// TwinCAT 3 PLC project PLC_TMO_VAC
// ProgramVersion: 3.1.4022.7
// libraries:
//   LCLS General, * (SLAC)
//   LCLS Vacuum, * (SLAC - LCLS)
//   PMPS, * (SLAC - LCLS)
//   Tc2_Standard, * (Beckhoff Automation GmbH)
//   Tc2_System, * (Beckhoff Automation GmbH)
//   Tc3_Module, * (Beckhoff Automation GmbH)
// project tree:
//   GVLs/ GVL_FEE_Device.TcGVL, GVL_PMPS.TcGVL, GVL_Variables.TcGVL
//   / PlcTask.TcTTO
//   POUs/ DIAGNOSTICS.TcPOU, MAIN.TcPOU, PRG_FEE.TcPOU, PRG_Section_2.TcPOU
// real-time tasks:
//   TASK PlcTask: cycle T#10ms, priority 20, ADS port 350
// I/O:
//   DEVICE Device 1 (EtherCAT), AmsNetId 5.59.117.180.2.1
//     B940-R20-CX0 (EK1200) [EK1200-5000 EtherCAT Power supply (2A E-Bus)]
//       CX0_E1 (EL2202)
//       CX0_E2 (EL1008)
//       CX0_E3 (EL2008)
//       CX0_E4 (EL2794)
//       CX0_E5 (EL6070)
//       CX0_E6_QPC1 (EL3064)
//       CX0_E7_QPC1 (EL1004)
//       CX0_E8_QPC1 (EL2794)
//       CX0_E9_QPC2 (EL3064)
//       CX0_E10_QPC2 (EL1004)
//       CX0_E11_QPC2 (EL2794)
//       CX0_E12 (EL6001)
//       EK1122-0080
//       EK (EL6692) [EL6692 EtherCAT Bridge terminal (Primary)]
//       CX0_EK1110
//     B940_R20_EK0 (EK1100) [EK1100 EtherCAT Coupler (2A E-Bus)]
//       Term 41 (EL3064)
//       Term 42 (EL3064)
//       Term 43 (EL2794)
//       Term 44 (EL9505)
//       Term 45 (EL1124)
//       Term 46 (EK1110)
//     B940_K4S20_EK0  (EK1100) [EK1100 EtherCAT Coupler (2A E-Bus)]
//       K420-E1-FSV (EL1004)
//       K420-E2-FSV (EL2202)
//       K420-E13-FSV (EL2202)
//       K420-E4-FSV (EK1110)
//     B940_K4S20_EB1  (EP2338-0002)
//     B940_K4S20_EB2  (EP3174-0002)
//     B940_K4S20_EB3 (EP2624-0002)
//     B940_K4S24_EB1 (EP3174-0002)
//     B940_K4S24_EB2 (EP2624-0002)
//     B940_K4S28_EB1 (EP3174-0002)
//     B940_K4S28_EB2 (EP2624-0002)
//     B940_K4S33_EB1 (EP2338-0002)
//     B940_K4S33_EB2 (EP3174-0002)
//     B940_K4S33_EB3 (EP2624-0002)
// variable links:
//   PLC_TMO_VAC Instance <-> Device 1 (EtherCAT)/B940-R20-CX0 (EK1200)/CX0_E10_QPC2 (EL1004)
//     PlcTask Inputs/GVL_FEE_Device.PC4K4_XTES_PIP_01.i_xSP_DI <-> Channel 1/Input
//   PLC_TMO_VAC Instance <-> Device 1 (EtherCAT)/B940-R20-CX0 (EK1200)/CX0_E11_QPC2 (EL2794)
//     PlcTask Outputs/GVL_FEE_Device.PC4K4_XTES_PIP_01.q_xHVEna_DO <-> Channel 1/Output
//   PLC_TMO_VAC Instance <-> Device 1 (EtherCAT)/B940-R20-CX0 (EK1200)/CX0_E6_QPC1 (EL3064)
//     PlcTask Inputs/GVL_FEE_Device.MR1K4_SOMS_PIP_01.i_iPRESS <-> AI Standard Channel 1/Value
//     PlcTask Inputs/GVL_FEE_Device.ST1K4_TEST_PIP_01.i_iPRESS <-> AI Standard Channel 2/Value
//     PlcTask Inputs/GVL_FEE_Device.ST2K4_BCS_PIP_01.i_iPRESS <-> AI Standard Channel 3/Value
//     PlcTask Inputs/GVL_FEE_Device.ST3K4_PPS_PIP_01.i_iPRESS <-> AI Standard Channel 4/Value
//   PLC_TMO_VAC Instance <-> Device 1 (EtherCAT)/B940-R20-CX0 (EK1200)/CX0_E7_QPC1 (EL1004)
//     PlcTask Inputs/GVL_FEE_Device.MR1K4_SOMS_PIP_01.i_xSP_DI <-> Channel 1/Input
//     PlcTask Inputs/GVL_FEE_Device.ST1K4_TEST_PIP_01.i_xSP_DI <-> Channel 2/Input
//     PlcTask Inputs/GVL_FEE_Device.ST2K4_BCS_PIP_01.i_xSP_DI <-> Channel 3/Input
//     PlcTask Inputs/GVL_FEE_Device.ST3K4_PPS_PIP_01.i_xSP_DI <-> Channel 4/Input
//   PLC_TMO_VAC Instance <-> Device 1 (EtherCAT)/B940-R20-CX0 (EK1200)/CX0_E8_QPC1 (EL2794)
//     PlcTask Outputs/GVL_FEE_Device.MR1K4_SOMS_PIP_01.q_xHVEna_DO <-> Channel 1/Output
//     PlcTask Outputs/GVL_FEE_Device.ST1K4_TEST_PIP_01.q_xHVEna_DO <-> Channel 2/Output
//     PlcTask Outputs/GVL_FEE_Device.ST2K4_BCS_PIP_01.q_xHVEna_DO <-> Channel 3/Output
//     PlcTask Outputs/GVL_FEE_Device.ST3K4_PPS_PIP_01.q_xHVEna_DO <-> Channel 4/Output
//   PLC_TMO_VAC Instance <-> Device 1 (EtherCAT)/B940-R20-CX0 (EK1200)/CX0_E9_QPC2 (EL3064)
//     PlcTask Inputs/GVL_FEE_Device.PC4K4_XTES_PIP_01.i_iPRESS <-> AI Standard Channel 1/Value
//   PLC_TMO_VAC Instance <-> Device 1 (EtherCAT)/B940_K4S20_EB1  (EP2338-0002)
//     PlcTask Inputs/GVL_FEE_Device.TV1K4_VGC_01.i_xClsLS <-> Channel 2/Input
//     PlcTask Inputs/GVL_FEE_Device.TV1K4_VGC_02.i_xClsLS <-> Channel 6/Input
//     PlcTask Inputs/GVL_FEE_Device.TV1K4_VGC_01.i_xOpnLS <-> Channel 1/Input
//     PlcTask Inputs/GVL_FEE_Device.TV1K4_VGC_02.i_xOpnLS <-> Channel 5/Input
//     PlcTask Outputs/GVL_FEE_Device.TV1K4_VGC_01.q_xOPN_DO <-> Channel 11/Output
//     PlcTask Outputs/GVL_FEE_Device.TV1K4_VGC_02.q_xOPN_DO <-> Channel 15/Output
//   PLC_TMO_VAC Instance <-> Device 1 (EtherCAT)/B940_K4S20_EB2  (EP3174-0002)
//     PlcTask Inputs/GVL_FEE_Device.TV1K4_GCC_01.i_iPRESS_R <-> AI Standard Channel 2/Value
//     PlcTask Inputs/GVL_FEE_Device.TV1K4_GPI_01.i_iPRESS_R <-> AI Standard Channel 1/Value
//   PLC_TMO_VAC Instance <-> Device 1 (EtherCAT)/B940_K4S20_EB3 (EP2624-0002)
//     PlcTask Outputs/GVL_FEE_Device.TV1K4_GCC_01.q_xHV_DIS <-> Channel 1/Output
//   PLC_TMO_VAC Instance <-> Device 1 (EtherCAT)/B940_K4S24_EB1 (EP3174-0002)
//     PlcTask Inputs/GVL_FEE_Device.ST1K4_TEST_GCC_01.i_iPRESS_R <-> AI Standard Channel 2/Value
//     PlcTask Inputs/GVL_FEE_Device.ST1K4_TEST_GPI_01.i_iPRESS_R <-> AI Standard Channel 1/Value
//   PLC_TMO_VAC Instance <-> Device 1 (EtherCAT)/B940_K4S24_EB2 (EP2624-0002)
//     PlcTask Outputs/GVL_FEE_Device.ST1K4_TEST_GCC_01.q_xHV_DIS <-> Channel 1/Output
//   PLC_TMO_VAC Instance <-> Device 1 (EtherCAT)/B940_K4S28_EB1 (EP3174-0002)
//     PlcTask Inputs/GVL_FEE_Device.ST2K4_BCS_GCC_01.i_iPRESS_R <-> AI Standard Channel 2/Value
//     PlcTask Inputs/GVL_FEE_Device.ST2K4_BCS_GPI_01.i_iPRESS_R <-> AI Standard Channel 1/Value
//   PLC_TMO_VAC Instance <-> Device 1 (EtherCAT)/B940_K4S28_EB2 (EP2624-0002)
//     PlcTask Outputs/GVL_FEE_Device.ST2K4_BCS_GCC_01.q_xHV_DIS <-> Channel 1/Output
//   PLC_TMO_VAC Instance <-> Device 1 (EtherCAT)/B940_K4S33_EB1 (EP2338-0002)
//     PlcTask Inputs/GVL_FEE_Device.ST3K4_PPS_VGC_01.i_xClsLS <-> Channel 2/Input
//     PlcTask Inputs/GVL_FEE_Device.ST3K4_PPS_VGC_01.i_xOpnLS <-> Channel 1/Input
//     PlcTask Outputs/GVL_FEE_Device.ST3K4_PPS_VGC_01.q_xOPN_DO <-> Channel 11/Output
//   PLC_TMO_VAC Instance <-> Device 1 (EtherCAT)/B940_K4S33_EB2 (EP3174-0002)
//     PlcTask Inputs/GVL_FEE_Device.PC4K4_XTES_GCC_01.i_iPRESS_R <-> AI Standard Channel 2/Value
//     PlcTask Inputs/GVL_FEE_Device.PC4K4_XTES_GPI_01.i_iPRESS_R <-> AI Standard Channel 1/Value
//   PLC_TMO_VAC Instance <-> Device 1 (EtherCAT)/B940_K4S33_EB3 (EP2624-0002)
//     PlcTask Outputs/GVL_FEE_Device.PC4K4_XTES_GCC_01.q_xHV_DIS <-> Channel 1/Output

CONFIGURATION PLC_TMO_VAC
    RESOURCE PLC ON TwinCAT3
        TASK PlcTask(INTERVAL := T#10ms, PRIORITY := 20);
        PROGRAM MAIN WITH PlcTask : MAIN;
    END_RESOURCE
END_CONFIGURATION

// ---- GVLs/GVL_FEE_Device.TcGVL
//{attribute 'qualified_only'}
VAR_GLOBAL




(* Isolation gate valves*)

	{attribute 'pytmc' :=' pv: TV1K4:VGC:01 '}
	{attribute 'TcLinkTo' := 	'.i_xOpnLS	:=	TIIB[B940_K4S20_EB1  (EP2338-0002)]^Channel 1^Input;
								 .i_xClsLS	:=	TIIB[B940_K4S20_EB1  (EP2338-0002)]^Channel 2^Input;
								.q_xOPN_DO	:=	TIIB[B940_K4S20_EB1  (EP2338-0002)]^Channel 11^Output'}
	TV1K4_VGC_01: FB_VGC;
	
	{attribute 'pytmc' :=' pv: TV1K4:VGC:02 '}
	{attribute 'TcLinkTo' := 	'.i_xOpnLS	:=	TIIB[B940_K4S20_EB1  (EP2338-0002)]^Channel 5^Input;
								 .i_xClsLS	:=	TIIB[B940_K4S20_EB1  (EP2338-0002)]^Channel 6^Input;
								 .q_xOPN_DO	:=	TIIB[B940_K4S20_EB1  (EP2338-0002)]^Channel 15^Output'}	
 	TV1K4_VGC_02: FB_VGC;

	{attribute 'pytmc' :=' pv: ST3K4:PPS:VGC:01 '}
	{attribute 'TcLinkTo' := 	'.i_xOpnLS	:=	TIIB[B940_K4S33_EB1 (EP2338-0002)]^Channel 1^Input;
								 .i_xClsLS	:=	TIIB[B940_K4S33_EB1 (EP2338-0002)]^Channel 2^Input;
								 .q_xOPN_DO	:=	TIIB[B940_K4S33_EB1 (EP2338-0002)]^Channel 11^Output'}	
	ST3K4_PPS_VGC_01 : FB_VGC;
	
(* Pirani & Cold Cathode*)

	(*Upstream Interface*)
	(*Gauges*)
	
	{attribute 'pytmc' :=' pv: MR1K4:GCC:01:ADS '}
//	(*MR1K4_GCC_01_ADS: FB_TGCC_ADS;*)
	MR1K4_GCC_01_ADS: FB_MKS500_EP;

	{attribute 'pytmc' :=' pv: TV1K4:GPI:01 '}
	{attribute 'TcLinkTo' := 	'.i_iPRESS_R	:=	TIIB[B940_K4S20_EB2  (EP3174-0002)]^AI Standard Channel 1^Value	'}
	TV1K4_GPI_01 : FB_MKS275;
	
	
	{attribute 'pytmc' :=' pv: TV1K4:GCC:01 '}
	{attribute 'TcLinkTo' := 	'.i_iPRESS_R	:=	TIIB[B940_K4S20_EB2  (EP3174-0002)]^AI Standard Channel 2^Value;
								 .q_xHV_DIS		:= 	TIIB[B940_K4S20_EB3 (EP2624-0002)]^Channel 1^Output	'}	
	TV1K4_GCC_01 : FB_MKS500_EP;
	
	{attribute 'pytmc' :=' pv: ST1K4:TEST:GPI:01 '}
	{attribute 'TcLinkTo' := 	'.i_iPRESS_R	:=	TIIB[B940_K4S24_EB1 (EP3174-0002)]^AI Standard Channel 1^Value		'}
	ST1K4_TEST_GPI_01 : FB_MKS275;
	
			
	{attribute 'pytmc' :=' pv: ST1K4:TEST:GCC:01 '}
	{attribute 'TcLinkTo' := 	'.i_iPRESS_R	:=	TIIB[B940_K4S24_EB1 (EP3174-0002)]^AI Standard Channel 2^Value;
								 .q_xHV_DIS		:= 	TIIB[B940_K4S24_EB2 (EP2624-0002)]^Channel 1^Output	'}	
	ST1K4_TEST_GCC_01 : FB_MKS500_EP;
	
	
	{attribute 'pytmc' :=' pv: ST2K4:BCS:GPI:01 '}
	{attribute 'TcLinkTo' := 	'.i_iPRESS_R	:=	TIIB[B940_K4S28_EB1 (EP3174-0002)]^AI Standard Channel 1^Value	'}
	ST2K4_BCS_GPI_01 : FB_MKS275;	
	
	{attribute 'pytmc' :=' pv: ST2K4:BCS:GCC:01 '}	
	{attribute 'TcLinkTo' := 	'.i_iPRESS_R	:=	TIIB[B940_K4S28_EB1 (EP3174-0002)]^AI Standard Channel 2^Value;
								 .q_xHV_DIS		:= 	TIIB[B940_K4S28_EB2 (EP2624-0002)]^Channel 1^Output	'}	
	ST2K4_BCS_GCC_01 : FB_MKS500_EP;		

						 
	{attribute 'pytmc' :=' pv: PC4K4:XTES:GPI:01 '}
	{attribute 'TcLinkTo' := 	'.i_iPRESS_R	:=	TIIB[B940_K4S33_EB2 (EP3174-0002)]^AI Standard Channel 1^Value	'}
	PC4K4_XTES_GPI_01 : FB_MKS275;

	{attribute 'pytmc' :=' pv: PC4K4:XTES:GCC:01 '}
	{attribute 'TcLinkTo' := 	'.i_iPRESS_R	:=	TIIB[B940_K4S33_EB2 (EP3174-0002)]^AI Standard Channel 2^Value;
								 .q_xHV_DIS		:= 	TIIB[B940_K4S33_EB3 (EP2624-0002)]^Channel 1^Output	'}	
	
	PC4K4_XTES_GCC_01 : FB_MKS500_EP;
	
	

	
(* Ion Pumps *)	
	
(*example
	{attribute 'TcLinkTo' := 	'.i_iPRESS		:=	TIIB[QPC_E1_EL3064]^AI Standard Channel 1^Value;
								 .i_xSP_DI		:= 	TIIB[QPC_E2_EL1004]^Channel 1^Input;
								 .q_xHVEna_DO	:= 	TIIB[QPC_E3_EL2794]^Channel 1^Output	'}
	{attribute 'pytmc' := '
		pv: RTDSL0:VAC:PIP:01
		io: io
	'}
	RTDSL0_PIP_01 : FB_PIP_Gamma;
	*)

	{attribute 'pytmc' :=' 
			pv: MR1K4:SOMS:PIP:01 '
 		}
	{attribute 'TcLinkTo' := 	'.i_iPRESS		:=	TIIB[CX0_E6_QPC1 (EL3064)]^AI Standard Channel 1^Value;
								 .i_xSP_DI		:= 	TIIB[CX0_E7_QPC1 (EL1004)]^Channel 1^Input;
								 .q_xHVEna_DO	:= 	TIIB[CX0_E8_QPC1 (EL2794)]^Channel 1^Output
	'}
	MR1K4_SOMS_PIP_01 : FB_PIP_Gamma;
	
	{attribute 'pytmc' :=' pv : ST1K4:TEST:PIP:01 '}
	{attribute 'TcLinkTo' := 	'.i_iPRESS		:=	TIIB[CX0_E6_QPC1 (EL3064)]^AI Standard Channel 2^Value;
								 .i_xSP_DI		:= 	TIIB[CX0_E7_QPC1 (EL1004)]^Channel 2^Input;
								 .q_xHVEna_DO	:= 	TIIB[CX0_E8_QPC1 (EL2794)]^Channel 2^Output
	'}	
	ST1K4_TEST_PIP_01 : FB_PIP_Gamma;	
	
	{attribute 'pytmc' :=' pv : ST2K4:BCS:PIP:01 '}
	{attribute 'TcLinkTo' := 	'.i_iPRESS		:=	TIIB[CX0_E6_QPC1 (EL3064)]^AI Standard Channel 3^Value;
								 .i_xSP_DI		:= 	TIIB[CX0_E7_QPC1 (EL1004)]^Channel 3^Input;
								 .q_xHVEna_DO	:= 	TIIB[CX0_E8_QPC1 (EL2794)]^Channel 3^Output
	'}
	ST2K4_BCS_PIP_01 : FB_PIP_Gamma;	

	{attribute 'pytmc' :=' pv : ST3K4:PPS:PIP:01 '}
	{attribute 'TcLinkTo' := 	'.i_iPRESS		:=	TIIB[CX0_E6_QPC1 (EL3064)]^AI Standard Channel 4^Value;
								 .i_xSP_DI		:= 	TIIB[CX0_E7_QPC1 (EL1004)]^Channel 4^Input;
								 .q_xHVEna_DO	:= 	TIIB[CX0_E8_QPC1 (EL2794)]^Channel 4^Output
	'}
	ST3K4_PPS_PIP_01 : FB_PIP_Gamma;		
	
	{attribute 'pytmc' :=' pv : PC4K4:XTES:PIP:01 '}
	{attribute 'TcLinkTo' := 	'.i_iPRESS		:=	TIIB[CX0_E9_QPC2 (EL3064)]^AI Standard Channel 1^Value;
								 .i_xSP_DI		:= 	TIIB[CX0_E10_QPC2 (EL1004)]^Channel 1^Input;
								 .q_xHVEna_DO	:= 	TIIB[CX0_E11_QPC2 (EL2794)]^Channel 1^Output
	'}
	PC4K4_XTES_PIP_01 : FB_PIP_Gamma;		

	
	
	

END_VAR

// ---- GVLs/GVL_PMPS.TcGVL
//{attribute 'qualified_only'}
VAR_GLOBAL
	
//Example implementation of the FFO
    {attribute 'pytmc' := '
    {pv: PLC:TMO:VAC:FF1    '}
    {attribute 'TcLinkTo' := '.q_xFastFaultOut:=TIIB[CX0_E1 (EL2202)]^Channel 1^Output'}
    g_FastFaultOutput1  :   FB_HardwareFFOutput;	//FFO for ST3K4_PPS's Upstream Components
	
	 {attribute 'pytmc' := 'pv: PLC:TMO:VAC:FF2  '}
    {attribute 'TcLinkTo' := '.q_xFastFaultOut:=TIIB[CX0_E1 (EL2202)]^Channel 2^Output'}
    g_FastFaultOutput2  :   FB_HardwareFFOutput;	//FFO for ST3K4_PPS's Downstream Components
	
	{attribute 'pytmc' := '    'pv: PLC:TMO:VAC:RESET:FF1    '}
	xReset_PMPS_FFO1	:	BOOL	:=	FALSE;		//FFO RESET for ST3K4_PPS's Upstream Components
	{attribute 'pytmc' := '    pv: PLC:TMO:VAC:RESET:FF2  '}
	xReset_PMPS_FFO2	:	BOOL	:=	FALSE;		//FFO RESET for ST3K4_PPS's Downstream Components
	
	
	xTMO_FEE_MPS_OK: BOOL := TRUE;
	
	xTMO_NEH_MPS_OK: BOOL := TRUE;

END_VAR

// ---- GVLs/GVL_Variables.TcGVL
//{attribute 'qualified_only'}
VAR_GLOBAL
	
	r_Accelerator_Setpoint	: REAL := 1E-12; (*unrealistic setpoint currently*)
	{attribute 'pytmc' := 'pv:VAC:OVRDON'}
//	xSystemOverrideMode_EBD	: BOOL := FALSE; (* Global system override for the HXR Vacuum System EBD*)
	xSystemOverrideMode_FEE	: BOOL := FALSE; (* Global system override for the HXR Vacuum System FEE*)
	xSystemOverrideMode_H1_1_H1_2	: BOOL := FALSE; (* Global system override for the HXR Vacuum System Hutch1.1 and Hutch1.2*)
END_VAR

// ---- POUs/MAIN.TcPOU
PROGRAM MAIN
VAR

//	fbLogHandler : FB_LogHandler;
	
END_VAR


//fbLogHandler();

// Run the Diagnostics PRG
DIAGNOSTICS();

(* FEE devices*)
PRG_FEE ();

END_PROGRAM

// ---- POUs/DIAGNOSTICS.TcPOU
PROGRAM DIAGNOSTICS
VAR
	//Change the PLC String Name to the actual PLC NAME
	sPLCName :STRING := 'PLC-LFE-VAC';
	//Link the sAMSNetID to the Etherat Master netID
	i_sAMSNetID AT %I*: AMSNETID;
	// DO NOT CHANGE
	sAMSNetID : STRING; //used for EPICS PV
	sLibVersion_LCLS_General : STRING;(* := stLibVersion_LCLS_General.sVersion*) ;
	fbEcatDiag:FB_EcatDiag;
	bAllSlaveStateGood : BOOL;
	bMasterStateGood :BOOL;
	iMasterState: WORD;
	sMasterState:STRING;
	nSlaveNumber : UINT;
	aiSlaveStates: ARRAY[1..256] OF BYTE;
	aEcSlaveInfo :  ARRAY[1..256] OF ST_EcDevice;
END_VAR

// Instaniating a call to the fbEcatDiag
fbEcatDiag(
	I_AMSNetId:=i_sAMSNetID , 
	i_xFirstPass:= _TaskInfo[1].FirstCycle, 
	q_xAllSlaveStatesGood=> bAllSlaveStateGood , 
	q_anTermStates=> aiSlaveStates, 
	q_xMasterStateGood=>bMasterStateGood , 
	q_nMasterState=> iMasterState, 
	q_sMasterState=> sMasterState , 
	q_astEcConfSlaveInfo=> aEcSlaveInfo , 
	q_nSlaves=> nSlaveNumber);

END_PROGRAM

// ---- POUs/PRG_FEE.TcPOU
PROGRAM PRG_FEE
VAR
ADS_connection_counter : UDINT;	
END_VAR

(* Gauges*)
   (* Read GCC from upstream PLC - plc-kfe-vac*)
  (* MR1K4_GCC_01_ADS(
	sNetId:= '172.21.92.61.1.1', 
	nPort:=851 , 
	sVarName:= 'fb_MR1K4_SOMS_GCC_1' , 
	iWatchdog:=ADS_connection_counter , 
	IG=> , 
	bError=> ); *)
	  

	TV1K4_GPI_01(); 
	ST1K4_TEST_GPI_01(); 
	ST2K4_BCS_GPI_01();
	PC4K4_XTES_GPI_01(); 
	
	TV1k4_GCC_01(PG:=TV1k4_GPI_01.PG , IG=> );
	ST1K4_TEST_GCC_01(PG:=ST1K4_TEST_GPI_01.PG , IG=> ); 
	ST2K4_BCS_GCC_01(PG:=ST2K4_BCS_GPI_01.PG , IG=> );
	PC4K4_XTES_GCC_01(PG:=PC4K4_XTES_GPI_01.PG , IG=> );
		
(* Valves*)
(*example
GEM1_VGC_10(i_stUSG := USG_GCC.IG, i_stDSG:= GEM1_GCC_10.IG,i_xDis_DPIlk := TRUE, i_xEPS_OK := TRUE,
		i_xPMPS_OK := TRUE, i_xExt_OK := xGEM1_AperturesOpnOK, i_xOverrideMode := xGEM1OverrideMode,i_xReset := xFastFaultReset,io_fbFFHWO :=g_FastFaultOutput1);
*)
	TV1K4_VGC_01(
				i_stUSG := MR1K4_GCC_01_ADS.IG, 
				i_stDSG:= TV1k4_GCC_01.IG, 
				i_xDis_DPIlk := FALSE, 
				i_xEPS_OK := TRUE,
				i_xPMPS_OK := TRUE, 
				i_xExt_OK := TRUE, 
				i_xOverrideMode := xSystemOverrideMode_FEE, 
				i_xReset := xReset_PMPS_FFO2,
				io_fbFFHWO :=g_FastFaultOutput1);
	
 	TV1K4_VGC_02(
				i_stUSG := TV1k4_GCC_01.IG, 
				i_stDSG:= ST1K4_TEST_GCC_01.IG, 
				i_xDis_DPIlk := FALSE, 
				i_xEPS_OK := TRUE,
				i_xPMPS_OK := TRUE, 
				i_xExt_OK := TRUE, 
				i_xOverrideMode := xSystemOverrideMode_FEE, 
				i_xReset := xReset_PMPS_FFO2,
				io_fbFFHWO :=g_FastFaultOutput1);
	
	ST3K4_PPS_VGC_01(
				i_stUSG := ST2K4_BCS_GCC_01.IG, 
				i_stDSG:= PC4K4_XTES_GCC_01.IG, 
				i_xDis_DPIlk := FALSE, 
				i_xEPS_OK := TRUE,
				i_xPMPS_OK := TRUE, 
				i_xExt_OK := TRUE, 
				i_xOverrideMode := xSystemOverrideMode_FEE, 
				i_xReset := xReset_PMPS_FFO2,
				io_fbFFHWO :=g_FastFaultOutput1);
				
(*Ion Pumps*)	
	(*example
	SP1L0_KMONO_PIP_01(i_stGauge:=SP1L0_KMONO_GCC_01.IG, stPump=>);*)		

	MR1K4_SOMS_PIP_01(i_stGauge := MR1K4_GCC_01_ADS.IG, stPump=>);
	ST1K4_TEST_PIP_01(i_stGauge := ST1K4_TEST_GCC_01.IG, stPump=>);
	ST2K4_BCS_PIP_01(i_stGauge := ST2K4_BCS_GCC_01.IG, stPump=>);
	ST3K4_PPS_PIP_01(i_stGauge := ST2K4_BCS_GCC_01.IG, stPump=>);
	PC4K4_XTES_PIP_01(i_stGauge := PC4K4_XTES_GCC_01.IG, stPump=>);

END_PROGRAM

// ---- POUs/PRG_Section_2.TcPOU
PROGRAM PRG_Section_2
VAR
END_VAR

END_PROGRAM
